PROGRAM POU_1
VAR
	T0: TOF;
	Te: TIME;
END_VAR

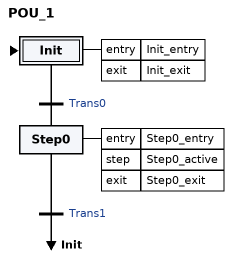
INITIAL_STEP Init:
    Init_entry(P1);  // entry action
    Init_exit(P0);  // exit action
END_STEP
TRANSITION FROM Init TO Step0
    := Trans0;
END_TRANSITION
STEP Step0:
    Step0_entry(P1);  // entry action
    Step0_active(N);  // step action
    Step0_exit(P0);  // exit action
END_STEP
TRANSITION FROM Step0 TO Init
    := Trans1;
END_TRANSITION

ACTION Init_entry:
Indicator.bSWGreen := TRUE;
SignalOut.bStart := TRUE;
END_ACTION

ACTION Init_exit:
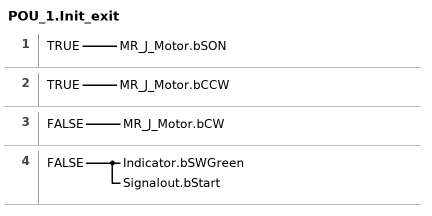
// NETWORK 1
MR_J_Motor.bSON := TRUE;

// NETWORK 2
MR_J_Motor.bCCW := TRUE;

// NETWORK 3
MR_J_Motor.bCW := FALSE;

// NETWORK 4
Indicator.bSWGreen := FALSE;
Signalout.bStart := FALSE;
END_ACTION

ACTION Step0_active:
Indicator.bSWGreen:=T0.Q;
Te := T0.ET;

IF Input.iHMISlide >= 0THEN
	MR_J_Motor.bCW := TRUE;
	MR_J_Motor.bCCW := FALSE;
ELSE
	MR_J_Motor.bCW := FALSE;
	MR_J_Motor.bCCW := TRUE;
END_IF
MR_J_Motor.iInVoltage := ABS(Input.iHMISlide);
END_ACTION

ACTION Step0_entry:
Indicator.bSWRed := TRUE;
END_ACTION

ACTION Step0_exit:
Indicator.bSWRed := FALSE;
MR_J_Motor.bSON := FALSE;
END_ACTION

TRANSITION Trans0:
Trans0:= (NOT Input.bSWGreen) AND Input.bEnable;
END_TRANSITION

TRANSITION Trans1:
Trans1 := (NOT Input.bSWRed) OR (NOT Input.bEMG);
END_TRANSITION

END_PROGRAM

(* stored: Version 1.1.0.1, ProductVersion 3.1.4026.6
   POU POU_1: Id {78c2347f-7356-4613-991f-414b53e8b4ef}, SpecialFunc None
   Action Init_entry: Id {b73c5e50-9444-43d8-823e-2fca70405876}
   Action Init_exit: Id {2cd803f4-7823-4636-afda-18721c3a6613}
   Action Step0_active: Id {aef13c31-31cf-4ce5-8fe3-c80e3befdabf}
   Action Step0_entry: Id {0eea0871-1a72-448f-885d-ff8ffc9253ad}
   Action Step0_exit: Id {f9db0f17-e146-4588-8acd-86f7223a3efe}
   Transition Trans0: Id {0e6cf033-9a07-4d6e-a728-2867995fe252}
   Transition Trans1: Id {03f62a7b-3d90-4359-ac9b-e874b9c2e9bb} *)
